(* CODESYS project TSR Libary.library
   Company: Eaton Automation
   Title: TSR Libary
   Description: Das ist eine Libary die die Wichtigsten Funktionen für den Touch-Simulations Roboter berteitstellt.
   Author: Samuel A. Marti
   Version: 0.80

Project tree, tasks and I/O mapping:
  libraries: Standard, 3.5.2.0 (System); CAA SerialCom, 3.5.3.0 (CAA Technical Workgroup)
  POUs/
    TSR Com/
      function block TSR_Com [ST]: A0_Start, A1_Get_Settings, A2_Open_Com, A3_Open_Wait, A4_Send_Com, A5_Send_Wait, A6_Receive_Com, A7_Receive_Wait, A8_String_Auswertung, A9_End, B100_Error
    FB Connect with TSR/
      function block Connect_with_TSR [ST]: A0_Start, A1_Progress, A2_Progress_Wait, A3_Auswerten, A4_End, B100_Error
    FN Set TSR startpoint/
      function FN_Set_TSR_startpoint [ST]
    FB Move TSR xy/
      function block FB_Move_TSR_xy [ST]: A0_Start, A1_Progress, A2_Progress_Wait, A3_Auswerten, A4_Wait_for_TSR, A5_Wait_for_TSR_Wait, A6_Wait_for_TSR_Auswerten, A7_End, B100_Error
    FB Go to TSR xy/
      function block FB_Go_to_TSR_xy [ST]: A0_Start, A1_Progress, A2_Progress_Wait, A3_Auswerten, A4_Wait_for_TSR, A5_Wait_for_TSR_Wait, A6_Wait_for_TSR_Auswerten, A7_End, B100_Error
    FB Get TSR position/
      function block FB_Get_TSR_position [ST]: A0_Start, A1_Progress, A2_Progress_Wait, A3_Auswerten, A4_End, B100_Error
    FB TSR Pen up down/
      function block TSR_Pen_up_down [ST]: A0_Start, A1_Progress, A2_Progress_Wait, A3_Auswerten, A4_End, B100_Error
  global variables GLOBAL
*)

// GLOBAL
VAR_GLOBAL
iStartPosx				:INT;			//Die Globale Variable des Neuen nulpunkts für die anderen FB's
iStartPosy				:INT;			//""
GTr_Faktor				:REAL := 8.8;	//Der umrechnungs Faktor: Momentan ist er auf mm abgestummen.
FB_TSRCom: 				TSR_Com;		//Die Com Communication
END_VAR

// POUs/TSR Com/TSR_Com
FUNCTION_BLOCK TSR_Com
VAR_INPUT
	xEXecute				:BOOL;		//Startbedingung für den FB.
	iCom					:INT;		//Die Nummer des Com Ports.
	stSendData				:STRING;	//Der String der Gesendet werden soll.
END_VAR

VAR_OUTPUT
	xBusy					:BOOL;		//Das Busy bit.
	xDone					:BOOL;		//Ist 1 wenn FB fertig ist.
	stReceivedData			:STRING;	//Der Empfangene Daten String.
	wState					:WORD;		//Der ENUM Wert für die ENUM Tabelle.
	xError					:BOOL;		//Ist 1 wenn es einen Error gab.
END_VAR

VAR
	LTi_Zustand				:INT;		//Der Zustand.
	LTi_PosString			:INT;		//Die Position vom Carisch retain lengfield.
	LTocpa_ComParameter1	:ARRAY[1..20] OF COM.PARAMETER; //Initalisierung der Com Parameter.
	
	LTx_ComOpen				:BOOL;		//Gibt an ob ein Com Port schon offen ist.
	LTudi_Handle			:UDINT;		//Der Interne COM Handle.
	LTst_ReceivedData		:STRING;	//Received Data zwischenspeicher.

	FB_ComOpen				:COM.Open;		//FB Open.
	FB_WriteCom				:Com.Write;		//FB Write.
	FB_ReadCom				:Com.Read;		//FB Read.
	FB_Timer				:TON;			//Timer Init
	
	GLRudi_ComPort			:UDINT;		//Welcher Com Port ist gemeint.
END_VAR


VAR CONSTANT
	GLRudi_StopBit			:UDINT := 0;	//Die Stopbits: 0 = 1stb, 1 = 1.5stb, 2 = 2stb.
	GLRudi_Parity			:UDINT := 2;	//Parity: 0 = gerade, 1 = ungerade, 2 = keine.
	GLRudi_Baudrate			:UDINT := 9600; //Möglich sind 2,5 m 115200 Bit/s, 5 m 57600 Bit/s, 10 m 38400 Bit/s, 15 m 19200 Bit/s, 30 m 9600 Bit/s
	GLRudi_TimeOut			:UDINT := 0;	//Keine ahnung was das bewirkt.
	GLRudi_BufferSize		:UDINT := 2048;	//Die Buffer grösse.
	GLRudi_ByteSize			:UDINT := 8;	//Die Grösse vom daten Byte. kann nur von 4 bis 8 sein
	GLRudi_Binary			:UDINT := 0;	//Binärmodus, keine EOF-Überprüfung/ keine ahnung wad das ist.
	GLRudi_OutxCTSFlow		:UDINT := 0;	//CTS Handshake auf Ausgang/ keine ahnung wad das ist.
	GLRudi_OutxDSRFlow		:UDINT := 0; 	//DSR Handshake auf Ausgang/ keine ahnung wad das ist.
	GLRudi_DTRControl		:UDINT := 0;	//DTR Control. DTR Flusssteuerung/ keine ahnung wad das ist.
	GLRudi_DSRSensitiv		:UDINT := 0; 	//DSR Empfindlichkeit/ keine ahnung wad das ist.
	GLRudi_RTSControl		:UDINT := 0;	//Rts Flussteuerung/ keine ahnung wad das ist.
	GLRudi_TXContinueOnXoff	:UDINT := 0;	//XOFF fortfahren Tx / keine ahnung wad das ist.
	GLRudi_OUTX				:UDINT := 0;	//XON/XOFF Ausgabeflusssteuerung / keine ahnung wad das ist.
	GLRudi_INX				:UDINT := 0;	//XON/XOFF Eingabeflusssteuerung / keine ahnung wad das ist.
	GLRudi_XOnChar			:UDINT := 0;	//Tx AND Rx XON Zeichen / keine ahnung wad das ist.
	GLRudi_XOffChar			:UDINT := 0;	//Tx AND Rx XOFF Zeichen.
	GLRudi_XOnLim			:UDINT := 0;	//Übertrage XON Schwellenwert
	GLRudi_XOffLim			:UDINT := 0;	//Übertrage XOFF Schwellenwert
	
	LTt_WaitTimeout		:TIME := T#2S;		//der Timout Timer.
	LTt_WaitCom			:TIME := T#600MS;	//Wait auf Received Data.
END_VAR

CASE LTi_Zustand OF
	0:
		A0_Start();					//Prüfe die Startbedingungen und Prüfe auf einen offenen Com Port
	1:
		A1_Get_Settings();			//Holt die Einstellungen für zu öffnenden Com Port.
	2:
		A2_Open_Com();				//Öffnet den Com Port.
	3:
		A3_Open_Wait();				//Wartet bis der Com Port offen ist.
	4:
		A4_Send_Com();				//Den String Senden.
	5:
		A5_Send_Wait();				//Warte bis der String gesendet wurde.
	6:
		A6_Receive_Com();			//Empfange den String.
	7:
		A7_Receive_Wait();			//Warte auf FB String lesen.
	8:
		A8_String_Auswertung();		//Werte den FB String aus.
	9:
		A9_End();					//Beende den FB vorgang und warte auf das zurücksetzten.
	100:
		B100_Error();				//Nur wenn ein Error gab.
END_CASE

FB_ComOpen();

ACTION A0_Start:
IF xExecute THEN			//Prüfe Startbedinung.
	xBusy := 1;				//Setze Busy.
	IF LTx_ComOpen THEN 	//Ist der Com Port offen ?
		LTi_Zustand := 4;	//Gehe direkt zum Schritt wo der String geschrieben wird.
	ELSE
		LTi_Zustand := 1;	//Gehe direkt zum Schritt wo der Com Port geöffnet wird.
	END_IF
END_IF
END_ACTION

ACTION A1_Get_Settings:
GLRudi_ComPort := INT_TO_UDINT(iCom);

//Port
LTocpa_ComParameter1[1].udiParameterId := COM.CAA_Parameter_Constants.udiPort;		//ID von Com Port
LTocpa_ComParameter1[1].udiValue := GLRudi_ComPort;									//Der COM Port1

//Stopbit
LTocpa_ComParameter1[2].udiParameterId := COM.CAA_Parameter_Constants.udiStopBits;	//ID von StopBit
LTocpa_ComParameter1[2].udiValue := GLRudi_StopBit;									//Der COM Port. 0 = 1stb, 1 = 1.5stb, 2 = 2stb.

//Parität
LTocpa_ComParameter1[3].udiParameterId := COM.CAA_Parameter_Constants.udiParity;		//ID von Parity
LTocpa_ComParameter1[3].udiValue := GLRudi_Parity;									//0 = gerade, 1 = ungerade, 2 = keine.

//Baudrate
LTocpa_ComParameter1[4].udiParameterId := COM.CAA_Parameter_Constants.udiBaudrate;	//ID von Baudrate
LTocpa_ComParameter1[4].udiValue := GLRudi_Baudrate;									//Möglich sind 2,5 m 115200 Bit/s, 5 m 57600 Bit/s, 10 m 38400 Bit/s, 15 m 19200 Bit/s, 30 m 9600 Bit/s

//Timeout
LTocpa_ComParameter1[5].udiParameterId := COM.CAA_Parameter_Constants.udiTimeout;	//ID von Timeout
LTocpa_ComParameter1[5].udiValue := GLRudi_TimeOut;									//Keine ahnung wad das ist.
(*
//BufferSize																		
LTocpa_ComParameter1[6].udiParameterId := COM.CAA_Parameter_Constants.udiBufferSize;	//ID von Buffersize
LTocpa_ComParameter1[6].udiValue := GLRudi_BufferSize;								//Die Grösse die der Buffer haben soll
*)
//ByteSize																	
LTocpa_ComParameter1[7].udiParameterId := COM.CAA_Parameter_Constants.udiByteSize;	//ID von ByteSize
LTocpa_ComParameter1[7].udiValue := GLRudi_ByteSize;									//Die Grösse vom daten Byte. kann nur von 4 bis 8 sein

//Binary
LTocpa_ComParameter1[8].udiParameterId := COM.CAA_Parameter_Constants.udiByteSize;	//ID von Binary
LTocpa_ComParameter1[8].udiValue := GLRudi_Binary;									//Binärmodus, keine EOF-Überprüfung/ keine ahnung wad das ist.
(*
//OutxCtsFlow
LTocpa_ComParameter1[9].udiParameterId := COM.CAA_Parameter_Constants.udiOutxCtsFlow;	//ID von OutxCtsFlow
LTocpa_ComParameter1[9].udiValue := GLRudi_OutxCTSFlow;									//CTS Handshake auf Ausgang/ keine ahnung wad das ist.

//OutxDSRFlow
LTocpa_ComParameter1[10].udiParameterId := COM.CAA_Parameter_Constants.udiOutxDsrFlow;	//ID von OutxDSRFlow
LTocpa_ComParameter1[10].udiValue := GLRudi_OutxDSRFlow;									//DSR Handshake auf Ausgang/ keine ahnung wad das ist.

//DTRControl
LTocpa_ComParameter1[11].udiParameterId := COM.CAA_Parameter_Constants.udiDtrControl;	//ID von DtrControl
LTocpa_ComParameter1[11].udiValue := GLRudi_OutxDSRFlow;									//DSR Handshake auf Ausgang/ keine ahnung wad das ist.

//DSR Sensitiv
LTocpa_ComParameter1[12].udiParameterId := COM.CAA_Parameter_Constants.udiDsrSensitivity;//ID von DSR Sensitiv
LTocpa_ComParameter1[12].udiValue := GLRudi_DSRSensitiv;									//DSR Empfindlichkeit/ keine ahnung wad das ist.

//RTS Control
LTocpa_ComParameter1[13].udiParameterId := COM.CAA_Parameter_Constants.udiRtsControl;	//ID von RTS Control
LTocpa_ComParameter1[13].udiValue := GLRudi_RTSControl;									//Rts Flusssteuerung/ keine ahnung wad das ist.

//TXContinueOnXoff	
LTocpa_ComParameter1[14].udiParameterId := COM.CAA_Parameter_Constants.udiTXContinueOnXoff;	//ID von  XOFF fortfahren Tx	
LTocpa_ComParameter1[14].udiValue := GLRudi_TXContinueOnXoff;									//XOFF fortfahren Tx / keine ahnung wad das ist.

//OUT X
LTocpa_ComParameter1[15].udiParameterId := COM.CAA_Parameter_Constants.udiOutX;	//ID von OUT X	
LTocpa_ComParameter1[15].udiValue := GLRudi_OUTX;									//XON/XOFF Ausgabeflusssteuerung/ keine ahnung wad das ist.

//IN X
LTocpa_ComParameter1[16].udiParameterId := COM.CAA_Parameter_Constants.udiInX;	//ID von IN X	
LTocpa_ComParameter1[16].udiValue := GLRudi_INX;									//Eingabeflusssteuerung/ keine ahnung wad das ist.

//XOnChar
LTocpa_ComParameter1[17].udiParameterId := COM.CAA_Parameter_Constants.udiXonChar;	//ID von x on char	
LTocpa_ComParameter1[17].udiValue := GLRudi_XOnChar;									//Tx AND Rx XON Zeichen/ keine ahnung wad das ist.

//XOffChar
LTocpa_ComParameter1[18].udiParameterId := COM.CAA_Parameter_Constants.udiXoffChar;	//ID von x off char
LTocpa_ComParameter1[18].udiValue := GLRudi_XOffChar;									//Tx AND Rx XOFF Zeichen/ keine ahnung wad das ist.

//XonLim
LTocpa_ComParameter1[19].udiParameterId := COM.CAA_Parameter_Constants.udiXonLim;	//ID von X on Lim
LTocpa_ComParameter1[19].udiValue := GLRudi_XOnLim;									//Übertrage XON Schwellenwert/ keine ahnung wad das ist.

//XoffLim
LTocpa_ComParameter1[20].udiParameterId := COM.CAA_Parameter_Constants.udiXonLim;	//ID von X off Lim
LTocpa_ComParameter1[20].udiValue := GLRudi_XOnLim;									//Übertrage XOFF Schwellenwert/ keine ahnung wad das ist.
*)
LTi_Zustand := 2;
END_ACTION

ACTION A2_Open_Com:
//Com Port öffnen
FB_ComOpen.usiListLength := SIZEOF(LTocpa_ComParameter1);	//Die länge der Parameter Liste
FB_ComOpen.pParameterList := ADR(LTocpa_ComParameter1);		//Die Adresse der Parameter Liste
FB_ComOpen.xExecute := 1;									//Start Flag setzten.
LTi_Zustand := 3;
FB_Timer(IN := 1, PT:= LTt_WaitTimeout);								//Rufe Timer auf
END_ACTION

ACTION A3_Open_Wait:
IF FB_ComOpen.xDone THEN											//Wenn der Port offen
	FB_Timer.IN := 0;					//Timer Zurücksetzten.
	LTi_Zustand := 4;					//Gehe in den Sende Schritt
	LTudi_Handle := FB_ComOpen.hCom;	//Speichere den Handle
	LTx_ComOpen	:= 1;					//Der Offene Com Port setzten.
ELSE
	IF FB_ComOpen.xError THEN				//Wenn es einen Error bei Com Port öffnen gab.
		FB_Timer.IN := 0;					//Timer Zurücksetzten.
		LTi_Zustand := 100;					//In den Error Zustand gehen.
		wState := 1;						//Den ENUM Wert Error angeben.
	ELSE
		IF FB_Timer.Q THEN						//Wenn der Timer Abgelaufen ist.
			LTi_Zustand := 100;					//In den Error Zustand gehen.
			wState := 4;						//Den ENUM Wert Error angeben.
			FB_Timer.IN := 0;
		END_IF
	END_IF
END_IF

FB_Timer();								//Rufe Timer auf
FB_ComOpen();							//Rufe den FB auf.
END_ACTION

ACTION A4_Send_Com:
FB_WriteCom(
	hCom			:= LTudi_Handle, 						//Ubergebe Handle.
	pBuffer 		:= ADR(stSendData),
	szSize 			:= INT_TO_UDINT(SIZEOF(stSendData)),
	xExecute		:= 1									//Starte Sende Vorgang.
);

LTi_Zustand := 5;
FB_Timer(IN := 1, PT:= LTt_WaitTimeout);				//Rufe Timer auf
END_ACTION

ACTION A5_Send_Wait:
IF FB_WriteCom.xDone THEN				//Wenn der String gesendet wurde.
	FB_Timer.IN := 0;					//Timer Zurücksetzten.
	LTi_Zustand := 6;					//Gehe in den Sende Schritt
ELSE
	IF FB_WriteCom.xError THEN				//Wenn es einen Error bei String senden gab.
		FB_Timer.IN := 0;					//Timer Zurücksetzten.
		LTi_Zustand := 100;					//In den Error Zustand gehen.
		wState := 2;						//Den ENUM Wert Error angeben.
	ELSE
		IF FB_Timer.Q THEN						//Wenn der Timer Abgelaufen ist.
			LTi_Zustand := 100;					//In den Error Zustand gehen.
			wState := 5;						//Den ENUM Wert Error angeben.
			FB_Timer.IN := 0;
		END_IF
	END_IF
END_IF

FB_Timer();								//Rufe Timer auf
FB_WriteCom();							//Rufe den FB auf.
END_ACTION

ACTION A6_Receive_Com:
FB_Timer(IN := 1, PT:= LTt_WaitCom);			//Rufe Timer auf
IF FB_TIMER.Q THEN							//Wenn der Timer fertig ist
	FB_Timer.IN := 0;						//Timer zurücksetzten
	FB_Timer();								//FB Timer zurückstzen.
	
	FB_ReadCom								//Rufe ReadCom auf.
	(
		xExecute	:= 1,					//Starte Lese STRING
		hCom		:= LTudi_Handle,		//übergib den Handle.
		pBuffer := ADR(LTst_ReceivedData),
		szBuffer := SIZEOF(LTst_ReceivedData),
	);
LTi_Zustand := 7;

END_IF
END_ACTION

ACTION A7_Receive_Wait:
IF FB_ReadCom.xDone THEN				//Wenn der String gesendet wurde.
	FB_Timer.IN := 0;					//Timer Zurücksetzten.
	LTi_Zustand := 8;					//Gehe in den Sende Schritt
ELSE
	IF FB_ReadCom.xError THEN				//Wenn es einen Error bei String senden gab.
		FB_Timer.IN := 0;					//Timer Zurücksetzten.
		LTi_Zustand := 100;					//In den Error Zustand gehen.
		wState := 3;						//Den ENUM Wert Error angeben.
	ELSE
		IF FB_Timer.Q THEN						//Wenn der Timer Abgelaufen ist.
			LTi_Zustand := 100;					//In den Error Zustand gehen.
			wState := 6;						//Den ENUM Wert Error angeben.
			FB_Timer.IN := 0;
		END_IF
	END_IF
FB_Timer(IN := 1, PT:= LTt_WaitTimeout);			//Schalte Timer ein.
END_IF

FB_Timer();								//Rufe Timer auf
FB_ReadCom();							//Rufe den FB auf.
END_ACTION

ACTION A8_String_Auswertung:
LTi_PosString := FIND(STR2:='$R$N' , STR1:=LTst_ReceivedData);		//Das caretsch Retain lengfield 
LTst_ReceivedData[LTi_PosString - 1] := 0;							//DAs caretain legas löschen mit allem was dahinter ist.
stReceivedData := LTst_ReceivedData;								//Ausgeben
LTi_Zustand := 9;													//Zum Zustand 9 gehen.
END_ACTION

ACTION A9_End:
xBusy := 0;							//Alles zurücksetzten
xDone := 1;
IF xExecute = 0 THEN				//Warten bis der User Zurückgesetzt hat.
	xDone := 0;
	LTi_Zustand := 0;
	stReceivedData := '';
	FB_WriteCom.xExecute := 0;
	FB_ReadCom.xExecute := 0;
	LTst_ReceivedData := '';
	FB_ComOpen.xExecute := 0;
	FB_WriteCom();
	FB_ReadCom();
	FB_ComOpen();
END_IF
END_ACTION

ACTION B100_Error:
xBusy := 0;							//Alles zurücksetzten
xError := 1;
IF xExecute = 0 THEN				//Wartem bis der User das xExecute zurückgesetzt hat.
	xError := 0;
	LTi_Zustand := 0;
	wState := 0;
	stReceivedData := '';
	LTst_ReceivedData := '';
	FB_WriteCom.xExecute := 0;
	FB_ReadCom.xExecute := 0;
	FB_ComOpen.xExecute := 0;
	FB_WriteCom();
	FB_ReadCom();
	FB_ComOpen();
END_IF
END_ACTION

END_FUNCTION_BLOCK

// POUs/FB Connect with TSR/Connect_with_TSR
FUNCTION_BLOCK Connect_with_TSR
VAR_INPUT
	xExecute				:BOOL;		//Startbedingung für den FB.
	iCom					:INT;		//Die Nummer des Com Ports.
END_VAR

VAR_OUTPUT
	xBusy					:BOOL;		//Das Busy bit.
	xDone					:BOOL;		//Ist 1 wenn FB fertig ist.
	wState					:WORD;		//Der ENUM Wert für die ENUM Tabelle.
	xError					:BOOL;		//Ist 1 wenn es einen Error gab.
END_VAR

VAR
	LTi_Zustand				:INT;		//Der Zustand.

	//TIMER
	FB_Timer				:TON;			//Timer Init
END_VAR

VAR CONSTANT
LTt_WaitTimeout		:TIME := T#2S;		//der Timout Timer.
END_VAR

CASE LTi_Zustand OF
	0:
		A0_Start();					//Prüfe die Startbedingungen 
	1:
		A1_Progress();				//Starte den Prozess.
	2:
		A2_Progress_Wait();			//Warte auf den FB TSR Com
	3:
		A3_Auswerten();				//Werte das Egebniss aus.
	4:
		A4_End();					//Warte auf Execute
	100:
		B100_Error();				//Nur wenn ein Error gab.
END_CASE

FB_TSRCom();

ACTION A0_Start:
IF xExecute THEN			//Prüfe Startbedinung.
	xBusy := 1;				//Setze Busy.
	LTi_Zustand := 1;	//Gehe direkt zum Schritt wo der Com Port geöffnet wird.
END_IF
END_ACTION

ACTION A1_Progress:
FB_TSRCom(						//TSR Com Aufrufen und Daten übergeben.
	xEXecute	:=	1 , 
	iCom		:= 	iCom, 
	stSendData	:= 	'?',  );
LTi_Zustand := 2;				//In den nächsten Zustand Wechseln.
END_ACTION

ACTION A2_Progress_Wait:
IF FB_TSRCom.xDone THEN											//Wenn der Port offen
	FB_Timer.IN := 0;					//Timer Zurücksetzten.
	LTi_Zustand := 3;					//Gehe in den Sende Schritt
ELSE
	IF FB_TSRCom.xError THEN				//Wenn es einen Error bei Com Port öffnen gab.
		FB_Timer.IN := 0;					//Timer Zurücksetzten.
		LTi_Zustand := 100;					//In den Error Zustand gehen.
		wState := FB_TSRCom.wState;			//Den ENUM Wert Error angeben.
	ELSE
		IF FB_Timer.Q THEN						//Wenn der Timer Abgelaufen ist.
			LTi_Zustand := 100;					//In den Error Zustand gehen.
			wState := 7;						//Den ENUM Wert Error angeben.
			FB_Timer.IN := 0;
		END_IF
	END_IF
FB_Timer(IN := 1, PT:= LTt_WaitTimeout);
END_IF

FB_Timer();								//Rufe Timer auf
END_ACTION

ACTION A3_Auswerten:
IF FB_TSRCom.stReceivedData = '!' THEN		//Wenn der TSR reagiert.
	LTi_Zustand := 4;						//Gehe zum letzten Zustand.
ELSE											
	LTi_Zustand := 100;	
	wState := 8;								
END_IF
END_ACTION

ACTION A4_End:
xBusy := 0;							//Alles zurücksetzten
xDone := 1;
IF xExecute = 0 THEN				//Warten bis der User Zurückgesetzt hat.
	xDone := 0;
	LTi_Zustand := 0;
	FB_TSRCom.xEXecute := 0;
END_IF
END_ACTION

ACTION B100_Error:
xBusy := 0;							//Alles zurücksetzten
xError := 1;
IF xExecute = 0 THEN				//Wartem bis der User das xExecute zurückgesetzt hat.
	xError := 0;
	LTi_Zustand := 0;
	wState := 0;
	FB_TSRCom.xEXecute := 0;
END_IF
END_ACTION

END_FUNCTION_BLOCK

// POUs/FN Set TSR startpoint/FN_Set_TSR_startpoint
FUNCTION FN_Set_TSR_startpoint : BOOL
VAR_INPUT
//FB EINGANGS VAR
iStartpointx			:INT;		//Der Virtuelle x Nullpunkt.
iStartpointy			:INT;		//Der Virtuelle y Nullpunkt.
END_VAR

iStartPosx := REAL_TO_INT(INT_TO_REAL(iStartpointx) * GTr_Faktor);		//Speicher eingang in Global Var
iStartPosy := REAL_TO_INT(INT_TO_REAL(iStartpointy) * GTr_Faktor);		//Speicher eingang in Global Var
FN_Set_TSR_startpoint := 1;		// Der Rückgabe wert der Funktion

END_FUNCTION

// POUs/FB Move TSR xy/FB_Move_TSR_xy
FUNCTION_BLOCK FB_Move_TSR_xy
VAR_INPUT
xExecute				:BOOL;		//Startbedingung für den FB.
iMovx					:INT;		//Die relative x bewegung des TSR in richtung x
iMovy					:INT;		//Die relative y bewegung des TSR in richtung y
END_VAR

VAR_OUTPUT
xBusy					:BOOL;		//Das Busy bit.
xDone					:BOOL;		//Ist 1 wenn FB fertig ist.
wState					:WORD;		//Der ENUM Wert für die ENUM Tabelle.
xError					:BOOL;		//Ist 1 wenn es einen Error gab.
END_VAR

VAR
LTi_Zustand				:INT;		//Der Zustand.
LTst_Zwischenspeicher	:STRING;	//Ein Zwischenspeicher für den Progress.
LTi_Len					:INT;		//Gibt die String länge an für den Progress.
LTi_x					:INT;		//Die x Schritte die der TSR machen soll.
LTi_y					:INT;		//Die y Schritte die der TSR machen soll.
//TIMER
FN_Timer				:TON;		//Timer Init.
END_VAR

//Parameters
VAR CONSTANT
LTt_WaitTimeout		:TIME := T#2S;		//der Timout Timer.
LTt_WaitCom			:TIME := T#250MS;	//Wait auf Received Data.
END_VAR

CASE LTi_Zustand OF
	0:
		A0_Start();						//Prüfe Startbedingunen
	1:
		A1_Progress();					//Starte den Prozess. und sende den Befehl an das TSR.
	2:
		A2_Progress_Wait();				//Warte auf den FB Com.
	3:
		A3_Auswerten();					//Beende den FB und warte auf den User.
	4:
		A4_Wait_for_TSR();				//Init warten bis der TSR bei der Position angekommen ist
	5:
		A5_Wait_for_TSR_Wait();			//Warte auf FB Com.
	6:
		A6_Wait_for_TSR_Auswerten();	//Werte aus.
	7:
		A7_End();						//Das ende der Funktion.
	100:
		B100_Error();					//Die Error Aktion.
END_CASE

FB_TSRCom();							//Aufrufen.

ACTION A0_Start:
IF xExecute THEN			//Prüfe Startbedinung.
	xBusy := 1;				//Setze Busy.
	LTi_Zustand := 1;		//nächster Schritt
END_IF
END_ACTION

ACTION A1_Progress:
//Hier wird der Befehl für den TSR zusammengesetzt.
LTst_Zwischenspeicher := 'mov ';	//Speicher

//Die Fakto miteinbeziehen so das die mm umgerechnet werden, in Schritte.
LTi_x := REAL_TO_INT(INT_TO_REAL(iMovx) * GTr_Faktor);
//Schreibe Die X koordinate hinein.
LTst_Zwischenspeicher := INSERT(LTst_Zwischenspeicher,INT_TO_STRING(LTi_x),4); 

//Finde die länge des String heraus
LTi_Len := LEN(STR := LTst_Zwischenspeicher);

//Schreibe am Schluss ein :
LTst_Zwischenspeicher := INSERT(LTst_Zwischenspeicher,':',LTi_Len);

//Die Fakto miteinbeziehen so das die mm umgerechnet werden, in Schritte.
LTi_y := REAL_TO_INT(INT_TO_REAL(iMovy) * GTr_Faktor);
//Nun schreibe hinter dem : die y Koordiante.
LTst_Zwischenspeicher := INSERT(LTst_Zwischenspeicher,INT_TO_STRING(LTi_y),(LTi_Len + 1));

//TSR Com Aufrufen und Daten übergeben.
FB_TSRCom(						
	iCom		:= 1,
	xEXecute	:=	1 , 
	stSendData	:= 	LTst_Zwischenspeicher,  );

//Auf zum nächsten schritt.
LTi_Zustand := 2;
END_ACTION

ACTION A2_Progress_Wait:
IF FB_TSRCom.xDone THEN											//Wenn der Port offen
	FN_Timer.IN := 0;						//Timer Zurücksetzten.
	LTi_Zustand := 3;						//Gehe in den Sende Schritt
ELSE
	IF FB_TSRCom.xError THEN				//Wenn es einen Error bei Com Port öffnen gab.
		FN_Timer.IN := 0;					//Timer Zurücksetzten.
		LTi_Zustand := 100;					//In den Error Zustand gehen.
		wState := FB_TSRCom.wState;			//Den ENUM Wert Error angeben.
	ELSE
		IF FN_Timer.Q THEN					//Wenn der Timer Abgelaufen ist.
			LTi_Zustand := 100;				//In den Error Zustand gehen.
			wState := 7;					//Den ENUM Wert Error angeben.
			FN_Timer.IN := 0;
		END_IF
	END_IF
FN_Timer(IN := 1, PT:= LTt_WaitTimeout);	//Setzte den Timer.
END_IF
FN_Timer();									//Timer Aufrufen.
END_ACTION

ACTION A3_Auswerten:
IF FB_TSRCom.stReceivedData = 'moving' THEN //Wenn der TSR reagiert.
	LTi_Zustand := 4;						//Gehe zum letzten Zustand.
	FB_TSRCom.xEXecute := 0;				//Setzte Com Communication zurück.
ELSE
	IF FB_TSRCom.stReceivedData = 'out of range' THEN
		wState := 9;						//out of range state
		LTi_zustand := 100;
	ELSE
		LTi_Zustand := 100;
		wState := 8;							//Gehe zum letzten Zustand.
	END_IF
END_IF
END_ACTION

ACTION A4_Wait_for_TSR:
//TSR Com Aufrufen und Daten übergeben.
FB_TSRCom(						
	iCom		:= 1,
	xEXecute	:=	1 , 
	stSendData	:= 'state',  );				//frage den Status ab.

//Auf zum nächsten schritt.
LTi_Zustand := 5;
END_ACTION

ACTION A5_Wait_for_TSR_Wait:
IF FB_TSRCom.xDone THEN											//Wenn der Port offen
	FN_Timer.IN := 0;						//Timer Zurücksetzten.
	LTi_Zustand := 6;						//Gehe in den Sende Schritt
ELSE
	IF FB_TSRCom.xError THEN				//Wenn es einen Error bei Com Port öffnen gab.
		FN_Timer.IN := 0;					//Timer Zurücksetzten.
		LTi_Zustand := 100;					//In den Error Zustand gehen.
		wState := FB_TSRCom.wState;			//Den ENUM Wert Error angeben.
	ELSE
		IF FN_Timer.Q THEN					//Wenn der Timer Abgelaufen ist.
			LTi_Zustand := 100;				//In den Error Zustand gehen.
			wState := 7;					//Den ENUM Wert Error angeben.
			FN_Timer.IN := 0;
		END_IF
	END_IF
FN_Timer(IN := 1, PT:= LTt_WaitTimeout);	//Setzte den Timer.
END_IF
FN_Timer();									//Timer Aufrufen.
END_ACTION

ACTION A6_Wait_for_TSR_Auswerten:
IF FB_TSRCom.stReceivedData = 'ready' THEN 		//Wenn der TSR reagiert.
	LTi_Zustand := 7;							//Gehe zum letzten Zustand.
	FB_TSRCom.xEXecute := 0;					//Setzte Com Communication zurück.
ELSE
	IF FB_TSRCom.stReceivedData = 'busy' THEN	//Wenn der TSR noch busy ist frage nochmal.
		FB_TSRCom.xEXecute := 0;				
		LTi_zustand := 4;
	ELSE
		IF FB_TSRCom.stReceivedData = '' THEN
			FB_TSRCom.xEXecute := 0;				
			LTi_zustand := 4;
		ELSE
			LTi_Zustand := 100;
			wState := 8;							//Gehe zum letzten Zustand.
		END_IF 
	END_IF
END_IF
END_ACTION

ACTION A7_End:
xBusy := 0;							//Alles zurücksetzten
xDone := 1;
IF xExecute = 0 THEN				//Warten bis der User Zurückgesetzt hat.
	xDone := 0;
	LTi_Zustand := 0;
	FB_TSRCom.xEXecute := 0;
END_IF
END_ACTION

ACTION B100_Error:
xBusy := 0;							//Alles zurücksetzten
xError := 1;
IF xExecute = 0 THEN				//Wartem bis der User das xExecute zurückgesetzt hat.
	xError := 0;
	LTi_Zustand := 0;
	wState := 0;					
	FB_TSRCom.xEXecute := 0;		//FB Com zurücksetzetn
END_IF
END_ACTION

END_FUNCTION_BLOCK

// POUs/FB Go to TSR xy/FB_Go_to_TSR_xy
FUNCTION_BLOCK FB_Go_to_TSR_xy
VAR_INPUT
xExecute				:BOOL;		//Startbedingung für den FB.
iGotox					:INT;		//Die relative x bewegung des TSR in richtung x
iGotoy					:INT;		//Die relative y bewegung des TSR in richtung y
END_VAR

VAR_OUTPUT
xBusy					:BOOL;		//Das Busy bit.
xDone					:BOOL;		//Ist 1 wenn FB fertig ist.
wState					:WORD;		//Der ENUM Wert für die ENUM Tabelle.
xError					:BOOL;		//Ist 1 wenn es einen Error gab.
END_VAR

VAR
LTi_Zustand				:INT;		//Der Zustand.
LTst_Zwischenspeicher	:STRING;	//Ein Zwischenspeicher für den Progress.
LTi_Len					:INT;		//Gibt die String länge an für den Progress.
LTi_x					:INT;		//Die x Schritte die der TSR machen soll.
LTi_y					:INT;		//Die y Schritte die der TSR machen soll.
//TIMER
FN_Timer				:TON;		//Timer Init.

END_VAR

//Parameters
VAR CONSTANT
LTt_WaitTimeout		:TIME := T#2S;		//der Timout Timer.
LTt_WaitCom			:TIME := T#250MS;	//Wait auf Received Data.
END_VAR

CASE LTi_Zustand OF
	0:
		A0_Start();						//Prüfe Startbedingunen
	1:
		A1_Progress();					//Starte den Prozess. und sende den Befehl an das TSR.
	2:
		A2_Progress_Wait();				//Warte auf den FB Com.
	3:
		A3_Auswerten();					//Beende den FB und warte auf den User.
	4:
		A4_Wait_for_TSR();				//Init warten bis der TSR bei der Position angekommen ist
	5:
		A5_Wait_for_TSR_Wait();			//Warte auf FB Com.
	6:
		A6_Wait_for_TSR_Auswerten();	//Werte aus.
	7:
		A7_End();						//Das ende der Funktion.
	100:
		B100_Error();					//Die Error Aktion.
END_CASE

FB_TSRCom();							//Aufrufen.

ACTION A0_Start:
IF xExecute THEN			//Prüfe Startbedinung.
	xBusy := 1;				//Setze Busy.
	LTi_Zustand := 1;		//nächster Schritt
END_IF
END_ACTION

ACTION A1_Progress:
//Hier wird der Befehl für den TSR zusammengesetzt.
LTst_Zwischenspeicher := 'movto ';	//Speicher

//Die Fakto miteinbeziehen so das die mm umgerechnet werden, in Schritte.
LTi_x := iStartPosx + (REAL_TO_INT(INT_TO_REAL(iGotox) * GTr_Faktor));
//Schreibe Die X koordinate hinein.
LTst_Zwischenspeicher := INSERT(LTst_Zwischenspeicher,INT_TO_STRING(LTi_x),6); 

//Finde die länge des String heraus
LTi_Len := LEN(STR := LTst_Zwischenspeicher);

//Schreibe am Schluss ein :
LTst_Zwischenspeicher := INSERT(LTst_Zwischenspeicher,':',LTi_Len);

//Die Fakto miteinbeziehen so das die mm umgerechnet werden, in Schritte.
LTi_y := iStartPosy + (REAL_TO_INT(INT_TO_REAL(iGotoy) * GTr_Faktor));
//Nun schreibe hinter dem : die y Koordiante.
LTst_Zwischenspeicher := INSERT(LTst_Zwischenspeicher,INT_TO_STRING(LTi_y),(LTi_Len + 1));

//TSR Com Aufrufen und Daten übergeben.
FB_TSRCom(						
	iCom		:= 1,
	xEXecute	:=	1 , 
	stSendData	:= 	LTst_Zwischenspeicher,  );

//Auf zum nächsten schritt.
LTi_Zustand := 2;
END_ACTION

ACTION A2_Progress_Wait:
IF FB_TSRCom.xDone THEN											//Wenn der Port offen
	FN_Timer.IN := 0;						//Timer Zurücksetzten.
	LTi_Zustand := 3;						//Gehe in den Sende Schritt
ELSE
	IF FB_TSRCom.xError THEN				//Wenn es einen Error bei Com Port öffnen gab.
		FN_Timer.IN := 0;					//Timer Zurücksetzten.
		LTi_Zustand := 100;					//In den Error Zustand gehen.
		wState := FB_TSRCom.wState;			//Den ENUM Wert Error angeben.
	ELSE
		IF FN_Timer.Q THEN					//Wenn der Timer Abgelaufen ist.
			LTi_Zustand := 100;				//In den Error Zustand gehen.
			wState := 7;					//Den ENUM Wert Error angeben.
			FN_Timer.IN := 0;
		END_IF
	END_IF
FN_Timer(IN := 1, PT:= LTt_WaitTimeout);	//Setzte den Timer.
END_IF
FN_Timer();									//Timer Aufrufen.
END_ACTION

ACTION A3_Auswerten:
IF FB_TSRCom.stReceivedData = 'moving' THEN //Wenn der TSR reagiert.
	LTi_Zustand := 4;						//Gehe zum letzten Zustand.
	FB_TSRCom.xEXecute := 0;				//Setzte Com Communication zurück.
ELSE
	IF FB_TSRCom.stReceivedData = 'out of range' THEN
		wState := 9;						//out of range state
		LTi_zustand := 100;
	ELSE
		LTi_Zustand := 100;
		wState := 8;							//Gehe zum letzten Zustand.
	END_IF
END_IF
END_ACTION

ACTION A4_Wait_for_TSR:
//TSR Com Aufrufen und Daten übergeben.
FB_TSRCom(						
	iCom		:= 1,
	xEXecute	:=	1 , 
	stSendData	:= 'state',  );				//frage den Status ab.

//Auf zum nächsten schritt.
LTi_Zustand := 5;
END_ACTION

ACTION A5_Wait_for_TSR_Wait:
IF FB_TSRCom.xDone THEN											//Wenn der Port offen
	FN_Timer.IN := 0;						//Timer Zurücksetzten.
	LTi_Zustand := 6;						//Gehe in den Sende Schritt
ELSE
	IF FB_TSRCom.xError THEN				//Wenn es einen Error bei Com Port öffnen gab.
		FN_Timer.IN := 0;					//Timer Zurücksetzten.
		LTi_Zustand := 100;					//In den Error Zustand gehen.
		wState := FB_TSRCom.wState;			//Den ENUM Wert Error angeben.
	ELSE
		IF FN_Timer.Q THEN					//Wenn der Timer Abgelaufen ist.
			LTi_Zustand := 100;				//In den Error Zustand gehen.
			wState := 7;					//Den ENUM Wert Error angeben.
			FN_Timer.IN := 0;
		END_IF
	END_IF
FN_Timer(IN := 1, PT:= LTt_WaitTimeout);	//Setzte den Timer.
END_IF
FN_Timer();									//Timer Aufrufen.
END_ACTION

ACTION A6_Wait_for_TSR_Auswerten:
IF FB_TSRCom.stReceivedData = 'ready' THEN 		//Wenn der TSR reagiert.
	LTi_Zustand := 7;							//Gehe zum letzten Zustand.
	FB_TSRCom.xEXecute := 0;					//Setzte Com Communication zurück.
ELSE
	IF FB_TSRCom.stReceivedData = 'busy' THEN	//Wenn der TSR noch busy ist frage nochmal.
		FB_TSRCom.xEXecute := 0;				
		LTi_zustand := 4;
	ELSE
		IF FB_TSRCom.stReceivedData = '' THEN
			FB_TSRCom.xEXecute := 0;				
			LTi_zustand := 4;
		ELSE
			LTi_Zustand := 100;
			wState := 8;							//Gehe zum letzten Zustand.
		END_IF 
	END_IF
END_IF
END_ACTION

ACTION A7_End:
xBusy := 0;							//Alles zurücksetzten
xDone := 1;
IF xExecute = 0 THEN				//Warten bis der User Zurückgesetzt hat.
	xDone := 0;
	LTi_Zustand := 0;
	FB_TSRCom.xEXecute := 0;
END_IF
END_ACTION

ACTION B100_Error:
xBusy := 0;							//Alles zurücksetzten
xError := 1;
IF xExecute = 0 THEN				//Wartem bis der User das xExecute zurückgesetzt hat.
	xError := 0;
	LTi_Zustand := 0;
	wState := 0;					
	FB_TSRCom.xEXecute := 0;		//FB Com zurücksetzetn
END_IF
END_ACTION

END_FUNCTION_BLOCK

// POUs/FB Get TSR position/FB_Get_TSR_position
FUNCTION_BLOCK FB_Get_TSR_position
VAR_INPUT
	//FB EINGANGS VAR
xExecute				:BOOL;		//Startbedingung für den FB.
END_VAR
VAR_OUTPUT
	//FB AUSGANGS VAR
xBusy					:BOOL;		//Das Busy bit.
xDone					:BOOL;		//Ist 1 wenn FB fertig ist.
wState					:WORD;		//Der ENUM Wert für die ENUM Tabelle.
xError					:BOOL;		//Ist 1 wenn es einen Error gab.
iPosx					:INT;		//Die Position vom TSR.
iPosy					:INT;		//Die Position vom TSR.
END_VAR

VAR
	//INTERNE VAR
LTi_Zustand				:INT;		//Der Zustand.
LTi_PosMid				:INT;		//Diese Variable soll angeben bei welcher Position sich das : vom rückgabe wert befindet.
LTi_Len					:INT;		//Gibt die String länge an für den Progress.
	
	//TIMER
FN_Timer				:TON;		//Timer Init.

END_VAR

//Parameters
VAR CONSTANT
LTt_WaitTimeout		:TIME := T#2S;		//der Timout Timer.
LTt_WaitCom			:TIME := T#250MS;	//Wait auf Received Data.
END_VAR

CASE LTi_Zustand OF
	0:
		A0_Start();					//Prüfe Startbedingunen
	1:
		A1_Progress();				//Starte den Prozess. und sende den Befehl an das TSR.
	2:
		A2_Progress_Wait();			//Warte auf den FB Com.
	3:
		A3_Auswerten();				//Beende den FB und warte auf den User.
	4:
		A4_End();					//Das ende der Funktion.
	100:
		B100_Error();				//Die Error Aktion.
END_CASE

FB_TSRCom();						//Aufrufen.

ACTION A0_Start:
IF xExecute THEN			//Prüfe Startbedinung.
	xBusy := 1;				//Setze Busy.
	LTi_Zustand := 1;		//nächster Schritt
END_IF
END_ACTION

ACTION A1_Progress:
//TSR Com Aufrufen und Daten übergeben.
FB_TSRCom(						
	iCom		:= 1,
	xEXecute	:= 1, 
	stSendData	:= 	'getpos',);

//Auf zum nächsten schritt.
LTi_Zustand := 2;
END_ACTION

ACTION A2_Progress_Wait:
IF FB_TSRCom.xDone THEN											//Wenn der Port offen
	FN_Timer.IN := 0;						//Timer Zurücksetzten.
	LTi_Zustand := 3;						//Gehe in den Sende Schritt
ELSE
	IF FB_TSRCom.xError THEN				//Wenn es einen Error bei Com Port öffnen gab.
		FN_Timer.IN := 0;					//Timer Zurücksetzten.
		LTi_Zustand := 100;					//In den Error Zustand gehen.
		wState := FB_TSRCom.wState;			//Den ENUM Wert Error angeben.
	ELSE
		IF FN_Timer.Q THEN					//Wenn der Timer Abgelaufen ist.
			LTi_Zustand := 100;				//In den Error Zustand gehen.
			wState := 7;					//Den ENUM Wert Error angeben.
			FN_Timer.IN := 0;
		END_IF
	END_IF
FN_Timer(IN := 1, PT:= LTt_WaitTimeout);	//Setzte den Timer.
END_IF
FN_Timer();									//Timer Aufrufen.
END_ACTION

ACTION A3_Auswerten:
LTi_PosMid := FIND(FB_TSRCom.stReceivedData,':');	//Speichert die Pos wo sich das : befindet.
LTi_Len	:=	LEN(FB_TSRCom.stReceivedData);
iPosx := REAL_TO_INT(INT_TO_REAL((STRING_TO_INT(LEFT(STR:=FB_TSRCom.stReceivedData , SIZE:=LTi_PosMid))) - iStartPosx) / GTr_Faktor);
iPosy := REAL_TO_INT(INT_TO_REAL((STRING_TO_INT(RIGHT(STR:=FB_TSRCom.stReceivedData , SIZE:=LTi_Len - LTi_PosMid))) - iStartPosy) / GTr_Faktor);
LTi_Zustand := 4;
END_ACTION

ACTION A4_End:
xBusy := 0;							//Alles zurücksetzten
xDone := 1;
IF xExecute = 0 THEN				//Warten bis der User Zurückgesetzt hat.
	xDone := 0;
	LTi_Zustand := 0;
	FB_TSRCom.xEXecute := 0;
	iPosx := 0;
	iPosy := 0;
END_IF
END_ACTION

ACTION B100_Error:
xBusy := 0;							//Alles zurücksetzten
xError := 1;
IF xExecute = 0 THEN				//Wartem bis der User das xExecute zurückgesetzt hat.
	xError := 0;
	LTi_Zustand := 0;
	wState := 0;					
	FB_TSRCom.xEXecute := 0;		//FB Com zurücksetzetn
	iPosx := 0;
	iPosy := 0;
END_IF
END_ACTION

END_FUNCTION_BLOCK

// POUs/FB TSR Pen up down/TSR_Pen_up_down
FUNCTION_BLOCK TSR_Pen_up_down
VAR_INPUT
	xExecute				:BOOL;		//Startbedingung für den FB.
	xPen					:BOOL;		//Wenn null = oben. und 1 = unten.
END_VAR

VAR_OUTPUT
	xBusy					:BOOL;		//Das Busy bit.
	xDone					:BOOL;		//Ist 1 wenn FB fertig ist.
	wState					:WORD;		//Der ENUM Wert für die ENUM Tabelle.
	xError					:BOOL;		//Ist 1 wenn es einen Error gab.
END_VAR

VAR
	LTi_Zustand				:INT;		//Der Zustand.
	LTst_String				:STRING;		//Ein Zwischenspeicher.
	//TIMER
	FB_Timer				:TON;			//Timer Init
END_VAR

VAR CONSTANT
LTt_WaitTimeout		:TIME := T#2S;		//der Timout Timer.
END_VAR

CASE LTi_Zustand OF
	0:
		A0_Start();					//Prüfe die Startbedingungen 
	1:
		A1_Progress();				//Starte den Prozess.
	2:
		A2_Progress_Wait();			//Warte auf den FB TSR Com
	3:
		A3_Auswerten();				//Werte das Egebniss aus.
	4:
		A4_End();					//Warte auf Execute
	100:
		B100_Error();				//Nur wenn ein Error gab.
END_CASE

FB_TSRCom();

ACTION A0_Start:
IF xExecute THEN			//Prüfe Startbedinung.
	xBusy := 1;				//Setze Busy.
	LTi_Zustand := 1;	//Gehe direkt zum Schritt wo der Com Port geöffnet wird.
END_IF
END_ACTION

ACTION A1_Progress:
IF xPen THEN
	LTst_String := 'touchdown';
ELSE
	LTst_String := 'touchup';
END_IF


FB_TSRCom(						//TSR Com Aufrufen und Daten übergeben.
	xEXecute	:=	1 ,  
	stSendData	:= 	LTst_String,  );
LTi_Zustand := 2;				//In den nächsten Zustand Wechseln.
END_ACTION

ACTION A2_Progress_Wait:
IF FB_TSRCom.xDone THEN											//Wenn der Port offen
	FB_Timer.IN := 0;					//Timer Zurücksetzten.
	LTi_Zustand := 3;					//Gehe in den Sende Schritt
ELSE
	IF FB_TSRCom.xError THEN				//Wenn es einen Error bei Com Port öffnen gab.
		FB_Timer.IN := 0;					//Timer Zurücksetzten.
		LTi_Zustand := 100;					//In den Error Zustand gehen.
		wState := FB_TSRCom.wState;			//Den ENUM Wert Error angeben.
	ELSE
		IF FB_Timer.Q THEN						//Wenn der Timer Abgelaufen ist.
			LTi_Zustand := 100;					//In den Error Zustand gehen.
			wState := 7;						//Den ENUM Wert Error angeben.
			FB_Timer.IN := 0;
		END_IF
	END_IF
FB_Timer(IN := 1, PT:= LTt_WaitTimeout);
END_IF

FB_Timer();								//Rufe Timer auf
END_ACTION

ACTION A3_Auswerten:
IF FB_TSRCom.stReceivedData = 'ok' THEN		//Wenn der TSR reagiert.
	LTi_Zustand := 4;						//Gehe zum letzten Zustand.
ELSE											
	LTi_Zustand := 100;	
	wState := 8;								
END_IF
END_ACTION

ACTION A4_End:
xBusy := 0;							//Alles zurücksetzten
xDone := 1;
IF xExecute = 0 THEN				//Warten bis der User Zurückgesetzt hat.
	xDone := 0;
	LTi_Zustand := 0;
	FB_TSRCom.xEXecute := 0;
END_IF
END_ACTION

ACTION B100_Error:
xBusy := 0;							//Alles zurücksetzten
xError := 1;
IF xExecute = 0 THEN				//Wartem bis der User das xExecute zurückgesetzt hat.
	xError := 0;
	LTi_Zustand := 0;
	wState := 0;
	FB_TSRCom.xEXecute := 0;
END_IF
END_ACTION

END_FUNCTION_BLOCK
